ABB RAPID module: mfc_rMach_path1.mod

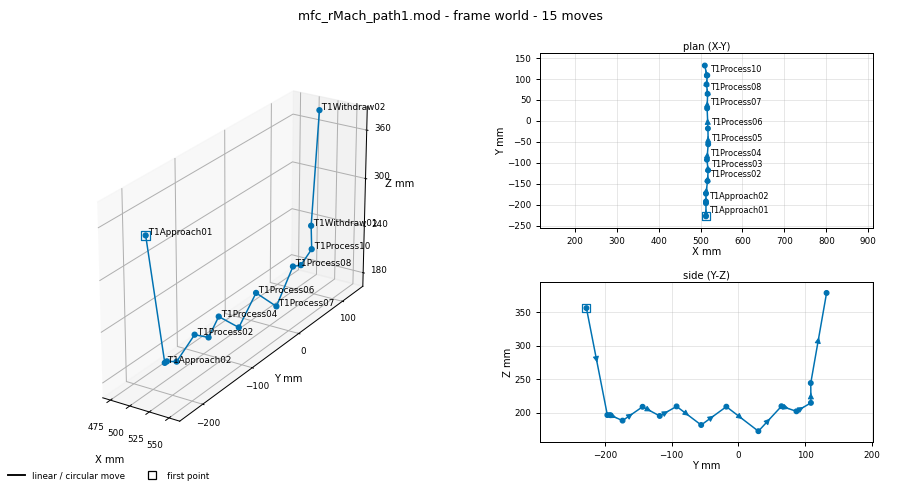
[picture p0: tool path of mfc_rMach_path1.mod in frame world, 15 of 15 moves have a stored position in this frame; points joined in program order, loops and branches not executed]
%%%
  VERSION: 1
  LANGUAGE: ENGLISH
%%%

MODULE mfc_rMach_path1

!This module is generated by RobotWare Machining FC V3.000. DO NOT EDIT.
!Any changes to this module will be lost when the RW Machining FC application is re-run and the program is exported.
LOCAL VAR robtarget T1Approach01 := [[513,-227.4,356.45],[0.000386385,0.796262,-0.604952,-0.000544438],[-1,-1,-2,0],[9E+09,9E+09,9E+09,9E+09,9E+09,9E+09]];
LOCAL VAR robtarget T1Approach02 := [[512.98,-196.06,196.29],[0.00038532,0.79626,-0.604955,-0.000537277],[-1,-1,-2,0],[9E+09,9E+09,9E+09,9E+09,9E+09,9E+09]];
LOCAL VAR robtarget T1Approach03 := [[512.97,-191.96,196.28],[0.000398504,0.796263,-0.604951,-0.000573975],[-1,-1,-2,0],[9E+09,9E+09,9E+09,9E+09,9E+09,9E+09]];
LOCAL VAR robtarget T1Approach04 := [[512.96,-173.29,187.97],[0.00039115,0.796256,-0.604959,-0.000550806],[-1,-1,-2,0],[9E+09,9E+09,9E+09,9E+09,9E+09,9E+09]];
LOCAL VAR robtarget T1Process01  := [[513.2,-172.81,187.96],[0.000534147,0.79621,-0.605019,-0.000968632],[-1,-1,-2,0],[9E+09,9E+09,9E+09,9E+09,9E+09,9E+09]];
LOCAL VAR robtarget T1Process02  := [[516.74,-143.31,208.7],[0.000553653,0.796489,-0.604652,-0.00085733],[-1,-1,-2,0],[9E+09,9E+09,9E+09,9E+09,9E+09,9E+09]];
LOCAL VAR robtarget T1Process03  := [[518.07,-117.61,194.93],[0.000624494,0.796442,-0.604714,-0.00094132],[-1,-1,-2,0],[9E+09,9E+09,9E+09,9E+09,9E+09,9E+09]];
LOCAL VAR robtarget T1Process04  := [[515.28,-92.42,209.25],[0.000342114,0.796222,-0.605004,-0.000346622],[-1,-1,-2,0],[9E+09,9E+09,9E+09,9E+09,9E+09,9E+09]];
LOCAL VAR robtarget T1Process05  := [[518.3,-55.59,181.39],[0.000601211,0.796412,-0.604754,-0.000803555],[-1,-1,-2,0],[9E+09,9E+09,9E+09,9E+09,9E+09,9E+09]];
LOCAL VAR robtarget T1Process06  := [[517.66,-17.89,208.86],[0.000659152,0.796497,-0.604641,-0.000869759],[-1,-1,-2,0],[9E+09,9E+09,9E+09,9E+09,9E+09,9E+09]];
LOCAL VAR robtarget T1Process07  := [[515.75,30.07,172.12],[0.000427854,0.796349,-0.604837,-0.000568856],[0,0,-2,0],[9E+09,9E+09,9E+09,9E+09,9E+09,9E+09]];
LOCAL VAR robtarget T1Process08  := [[516.9,64.62,209.49],[0.00072138,0.7966,-0.604506,-0.000814757],[0,0,-2,0],[9E+09,9E+09,9E+09,9E+09,9E+09,9E+09]];
LOCAL VAR robtarget T1Process09  := [[514.36,87.06,201.9],[0.000977252,0.796579,-0.604533,-0.000988229],[0,0,-2,0],[9E+09,9E+09,9E+09,9E+09,9E+09,9E+09]];
LOCAL VAR robtarget T1Process10  := [[516.13,108.71,214.53],[0.000720287,0.796691,-0.604386,-0.000705827],[0,0,-2,0],[9E+09,9E+09,9E+09,9E+09,9E+09,9E+09]];
LOCAL VAR robtarget T1Withdraw01 := [[515.07,108.5,244.22],[0.000427521,0.796683,-0.604397,-0.000457166],[0,0,-2,0],[9E+09,9E+09,9E+09,9E+09,9E+09,9E+09]];
LOCAL VAR robtarget T1Withdraw02 := [[510.21,132.17,379.13],[0.000495201,0.796668,-0.604417,-0.000501833],[0,0,-2,0],[9E+09,9E+09,9E+09,9E+09,9E+09,9E+09]];
LOCAL VAR num n1ForceX := 0;
LOCAL VAR num n1ForceY := 0;
LOCAL VAR num n1ForceZ := -10;


PROC run_rMach_path1 (bool bRecover, bool bSpindleOn)
	FCDeact;

	IF bRecover = true THEN
		FCCalib  tool0_LD \Recovery;
	ELSE
		FCCalib  tool0_LD;
	ENDIF

	IF bSpindleOn = true THEN
		SpindleOn;
	ENDIF

	MoveL T1Approach01, v50, z1,tool0\wobj :=wobj0;
	MoveL T1Approach02, v50, z1,tool0\wobj :=wobj0;
	MoveL T1Approach03, v50, z1,tool0\wobj :=wobj0;
	MoveL T1Approach04, v50, fine,tool0\wobj :=wobj0;

	FCPress1LStart T1Process01, v50 \Fx:= n1ForceX \Fy:= n1ForceY \Fz:= n1ForceZ,50 \ForceFrameRef:=FC_REFFRAME_TOOL \ForceChange:=50 \DampingTune:=100 \TimeOut:=5, \UseSpdFFW, \PosSupvDist:=9e9, z1, tool0 \wobj:=wobj0;
	FCPressL T1Process02, v50, 10, z1, tool0, \wobj:=wobj0;
	FCPressL T1Process03, v50, 10, z1, tool0, \wobj:=wobj0;
	FCPressL T1Process04, v50, 10, z1, tool0, \wobj:=wobj0;
	FCPressL T1Process05, v50, 10, z1, tool0, \wobj:=wobj0;
	FCPressL T1Process06, v50, 10, z1, tool0, \wobj:=wobj0;
	FCPressL T1Process07, v50, 10, z1, tool0, \wobj:=wobj0;
	FCPressL T1Process08, v50, 10, z1, tool0, \wobj:=wobj0;
	FCPressL T1Process09, v50, 10, z1, tool0, \wobj:=wobj0;
	FCPressL T1Process10, v50, 10, z1, tool0, \wobj:=wobj0;

	FCPressLEnd T1Withdraw01,v50,\ForceChange :=50,\ZeroContactValue := 5;
	MoveL T1Withdraw02, v50, z1,tool0\wobj :=wobj0;

	IF bSpindleOn = true THEN
		SpindleOff;
	ENDIF

ENDPROC

ENDMODULE
